{attribute 'qualified_only'}
{attribute 'strict'}
TYPE E_ServoTypeMoves :
(
	AbsoluteMove := 0,
	RelativeMove := 1,
	VelocityMove := 2,
	DynamicGear  := 3
);
END_TYPE

(* stored: Version 1.1.0.1, ProductVersion 3.1.4024.12
   DUT E_ServoTypeMoves: Id {c73a34db-063f-4e6d-825e-1c756e9acd05} *)
